{attribute 'GeneratedUsingTerminal: KL6211-0020'}
{attribute addProperty BoxType "KL6211-0020"}
{attribute addProperty Id "StatusAT %I*UINT0Parameter_InAT %I*UDINT0ASI_In_StatusAT %I*BYTE0ASI_In_Slave_1AT %I*BYTE0ASI_In_Slave_2AT %I*BYTE0ASI_In_Slave_3AT %I*BYTE0ASI_In_Slave_4AT %I*BYTE0ASI_In_Slave_5AT %I*BYTE0ASI_In_Slave_6AT %I*BYTE0ASI_In_Slave_7AT %I*BYTE0ASI_In_Slave_8AT %I*BYTE0ASI_In_Slave_9AT %I*BYTE0ASI_In_Slave_10AT %I*BYTE0ASI_In_Slave_11AT %I*BYTE0ControlAT %Q*UINT0Parameter_OutAT %Q*UDINT0ASI_Out_ControlAT %Q*BYTE0ASI_Out_Slave_1AT %Q*BYTE0ASI_Out_Slave_2AT %Q*BYTE0ASI_Out_Slave_3AT %Q*BYTE0ASI_Out_Slave_4AT %Q*BYTE0ASI_Out_Slave_5AT %Q*BYTE0ASI_Out_Slave_6AT %Q*BYTE0ASI_Out_Slave_7AT %Q*BYTE0ASI_Out_Slave_8AT %Q*BYTE0ASI_Out_Slave_9AT %Q*BYTE0ASI_Out_Slave_10AT %Q*BYTE0ASI_Out_Slave_11AT %Q*BYTE0"}
{attribute addProperty CRC "161205466"}
{attribute addProperty Size "0"}
TYPE Channel_099BCCDA :
STRUCT
	{attribute addProperty Name "Status"}
	Status AT %I* : UINT;
	{attribute addProperty Name "Parameter_In"}
	Parameter_In AT %I* : UDINT;
	{attribute addProperty Name "ASI_In_Status"}
	ASI_In_Status AT %I* : BYTE;
	{attribute addProperty Name "ASI_In_Slave_1"}
	ASI_In_Slave_1 AT %I* : BYTE;
	{attribute addProperty Name "ASI_In_Slave_2"}
	ASI_In_Slave_2 AT %I* : BYTE;
	{attribute addProperty Name "ASI_In_Slave_3"}
	ASI_In_Slave_3 AT %I* : BYTE;
	{attribute addProperty Name "ASI_In_Slave_4"}
	ASI_In_Slave_4 AT %I* : BYTE;
	{attribute addProperty Name "ASI_In_Slave_5"}
	ASI_In_Slave_5 AT %I* : BYTE;
	{attribute addProperty Name "ASI_In_Slave_6"}
	ASI_In_Slave_6 AT %I* : BYTE;
	{attribute addProperty Name "ASI_In_Slave_7"}
	ASI_In_Slave_7 AT %I* : BYTE;
	{attribute addProperty Name "ASI_In_Slave_8"}
	ASI_In_Slave_8 AT %I* : BYTE;
	{attribute addProperty Name "ASI_In_Slave_9"}
	ASI_In_Slave_9 AT %I* : BYTE;
	{attribute addProperty Name "ASI_In_Slave_10"}
	ASI_In_Slave_10 AT %I* : BYTE;
	{attribute addProperty Name "ASI_In_Slave_11"}
	ASI_In_Slave_11 AT %I* : BYTE;
	{attribute addProperty Name "Control"}
	Control AT %Q* : UINT;
	{attribute addProperty Name "Parameter_Out"}
	Parameter_Out AT %Q* : UDINT;
	{attribute addProperty Name "ASI_Out_Control"}
	ASI_Out_Control AT %Q* : BYTE;
	{attribute addProperty Name "ASI_Out_Slave_1"}
	ASI_Out_Slave_1 AT %Q* : BYTE;
	{attribute addProperty Name "ASI_Out_Slave_2"}
	ASI_Out_Slave_2 AT %Q* : BYTE;
	{attribute addProperty Name "ASI_Out_Slave_3"}
	ASI_Out_Slave_3 AT %Q* : BYTE;
	{attribute addProperty Name "ASI_Out_Slave_4"}
	ASI_Out_Slave_4 AT %Q* : BYTE;
	{attribute addProperty Name "ASI_Out_Slave_5"}
	ASI_Out_Slave_5 AT %Q* : BYTE;
	{attribute addProperty Name "ASI_Out_Slave_6"}
	ASI_Out_Slave_6 AT %Q* : BYTE;
	{attribute addProperty Name "ASI_Out_Slave_7"}
	ASI_Out_Slave_7 AT %Q* : BYTE;
	{attribute addProperty Name "ASI_Out_Slave_8"}
	ASI_Out_Slave_8 AT %Q* : BYTE;
	{attribute addProperty Name "ASI_Out_Slave_9"}
	ASI_Out_Slave_9 AT %Q* : BYTE;
	{attribute addProperty Name "ASI_Out_Slave_10"}
	ASI_Out_Slave_10 AT %Q* : BYTE;
	{attribute addProperty Name "ASI_Out_Slave_11"}
	ASI_Out_Slave_11 AT %Q* : BYTE;
END_STRUCT
END_TYPE

(* stored: Version 1.2.0.0, ProductVersion 3.1.4024.9
   DUT Channel_099BCCDA: Id {50790d3d-321a-4d07-8424-5bc786578d52} *)
